TYPE ST_St010_IO_IN :
STRUCT	
	// inputs
	bRefpos	: BOOL;	// Sensor | Oven | Referenzposition | BMK: =P260+xyz- | Terminal: .: | Tc3Hmi
	
END_STRUCT
END_TYPE

(* stored: Version 1.1.0.1
   DUT ST_St010_IO_IN: Id {076c8679-defe-4c73-a920-c9ab0eb70958} *)
